// TIA Portal project "test_web_ 3" (V15)

(* hardware
DEVICE "S7-1200 station_1"  S7-1200 Station
   slot 0: "Rack_0"  S7-1200 Rack  Rack  V1.0
   slot 1: "PLC_1"  CPU 1214C DC/DC/DC  6ES7 214-1AG40-0XB0  V4.2
   slot 2: "DQ 16x24VDC_1"  SM 1222 DQ16 x 24VDC  6ES7 222-1BH32-0XB0  V2.0
*)

// ===== PLC "PLC_1"  CPU 1214C DC/DC/DC =====

VAR_GLOBAL   // PLC tag table "Default tag table"
   "System_Byte" AT %MB1 : Byte;
   "FirstScan" AT %M1.0 : Bool;
   "DiagStatusUpdate" AT %M1.1 : Bool;
   "AlwaysTRUE" AT %M1.2 : Bool;
   "AlwaysFALSE" AT %M1.3 : Bool;
   "Clock_Byte" AT %MB0 : Byte;
   "Clock_10Hz" AT %M0.0 : Bool;
   "Clock_5Hz" AT %M0.1 : Bool;
   "Clock_2.5Hz" AT %M0.2 : Bool;
   "Clock_2Hz" AT %M0.3 : Bool;
   "Clock_1.25Hz" AT %M0.4 : Bool;
   "Clock_1Hz" AT %M0.5 : Bool;
   "Clock_0.625Hz" AT %M0.6 : Bool;
   "Clock_0.5Hz" AT %M0.7 : Bool;
   "Tag_1" AT %MW0 : Int;
   "Tag_2" AT %MW10 : Int;
   "Tag_3" AT %M100.0 : Bool;
   "Tag_4" AT %M100.1 : Bool;
END_VAR

VAR_GLOBAL   // PLC tag table "output"
   "q0.4" AT %Q0.4 : Bool;
END_VAR

DATA_BLOCK "WEB_COM"   // DB1
{ S7_Optimized_Access := 'TRUE' }
VERSION : 0.1
   VAR
      tag_bool : Bool;
      tag_int : Int;
      tag_byte : Byte;
      tag_real : Real;
      tag_string : String;
      tag_int_2 : Int;
      Start : Bool;
      Stop : Bool;
      Data6 : DWord;
      Data5 : Real;
      Data1 : Int;
      Data4 : Int;
      Data3 : DInt;
      Data2 : Real;
      Static_1 : Int;
   END_VAR
BEGIN
END_DATA_BLOCK

// folder: System blocks/Program resources

DATA_BLOCK "IEC_Counter_0_DB"   // DB2
{ S7_Optimized_Access := 'TRUE' }
AUTHOR : Simatic
FAMILY : IEC
NAME : CNTR
VERSION : 1.0
// stored: InstanceOfName IEC_COUNTER
"IEC_COUNTER"
BEGIN
END_DATA_BLOCK

DATA_BLOCK "IEC_Counter_0_DB_1"   // DB3
{ S7_Optimized_Access := 'TRUE' }
AUTHOR : Simatic
FAMILY : IEC
NAME : CNTR
VERSION : 1.0
// stored: InstanceOfName IEC_COUNTER
"IEC_COUNTER"
BEGIN
END_DATA_BLOCK

// folder: (top level)

ORGANIZATION_BLOCK "Main"   // OB1, LAD, ProgramCycle
TITLE = "Main Program Sweep (Cycle)"
{ S7_Optimized_Access := 'TRUE' }
VERSION : 0.1
   VAR_INPUT
      Initial_Call : Bool;   // Initial call of this OB
      Remanence : Bool;   // =True, if remanent data are available
   END_VAR
   VAR_TEMP   // added for the SCL form of the ladder/FBD networks
      _w1 : Bool;
   END_VAR
BEGIN

REGION Network 1
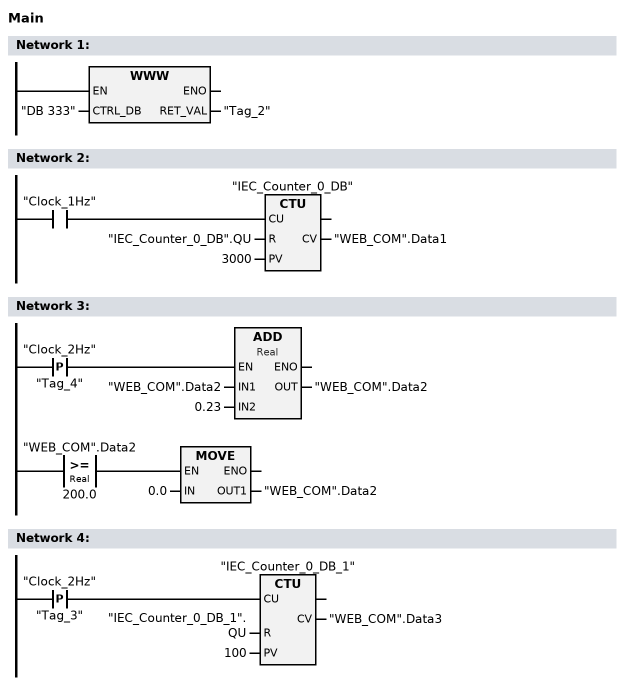
   "Tag_2" := WWW(CTRL_DB := "DB 333");
END_REGION

REGION Network 2
   "IEC_Counter_0_DB".CTU(CU := "Clock_1Hz", R := "IEC_Counter_0_DB".QU, PV := 3000, CV => "WEB_COM".Data1);
END_REGION

REGION Network 3
   RUNG wire#powerrail
      P_Contact(operand := "Clock_2Hz", bit := "Tag_4")
      { S7_Templates := "SrcType := Real" } Add(in1 := "WEB_COM".Data2, in2 := 0.23, out => "WEB_COM".Data2)
   END_RUNG
   RUNG wire#powerrail
      { S7_Templates := "SrcType := Real" } GE_Contact(in1 := "WEB_COM".Data2, in2 := 200.0)
      Move(in := 0.0, out1 => "WEB_COM".Data2)
   END_RUNG
   // the same network as SCL:
   #_w1 := "Clock_2Hz" AND NOT "Tag_4";   // rising edge of "Clock_2Hz"
   "Tag_4" := "Clock_2Hz";
   IF #_w1 THEN "WEB_COM".Data2 := "WEB_COM".Data2 + 0.23; END_IF;
   IF "WEB_COM".Data2 >= 200.0 THEN "WEB_COM".Data2 := 0.0; END_IF;
END_REGION

REGION Network 4
   #_w1 := "Clock_2Hz" AND NOT "Tag_3";   // rising edge of "Clock_2Hz"
   "Tag_3" := "Clock_2Hz";
   "IEC_Counter_0_DB_1".CTU(CU := #_w1, R := "IEC_Counter_0_DB_1".QU, PV := 100, CV => "WEB_COM".Data3);
END_REGION
END_ORGANIZATION_BLOCK